PROGRAM MAIN_ST03
VAR
	fbStation03							: RACBaseObjects.FB_Station;
END_VAR

fbStation03(bInitFinished := FALSE);

END_PROGRAM

(* stored: Version 1.1.0.1, ProductVersion 3.1.4024.12
   POU MAIN_ST03: Id {dc3e1128-42a6-4adf-9d15-fe50aa910b74}, SpecialFunc None *)
